FUNCTION_BLOCK FB_EQ2HOR2
VAR_INPUT
	// right ascension in degrees
	alpha: LREAL;
	// declination in degrees
	delta: LREAL;
	// longitude in degrees
	lon: LREAL;
	// latitude in degrees
	lat: LREAL;
	// Julian Days
	JD: LREAL;
END_VAR
VAR_OUTPUT
	// altitude in degrees
	alt: LREAL;
	// azimuth in degrees
	az: LREAL;
	// hour angle in degreesss
	ha: LREAL;
END_VAR
VAR
	lst: LREAL;
	// helper variables
	sinalt, sinaz, cosaz, cosalt, az1, az2, az3, length,
	// in radians
	phi_r, tau_r, alpha_r, delta_r: LREAL;
	// current epoch
	J_now: 		LREAL;
	// enable precession
	precess: 	BOOL := TRUE;
	// precession function block
	fbprecess: 	FB_PRECESS;
	//precessed coordinates
	alpha1, delta1:	LREAL;
END_VAR
VAR CONSTANT
	d2r:	LREAL := PI/180.0;
	r2d:	LREAL := 180.0/PI;
	//h2r:	LREAL := PI/12.0;
	//h2d:	LREAL := 15.0;
END_VAR

(* 
source: http://star-www.st-and.ac.uk/~fv/webnotes/chapter7.htm
https://squarewidget.com/astronomical-calculations-sidereal-time/

*)
lst := ct2lst(lon, jd) * 15.0; // lst in degrees

J_now := (JD - 2451545.0)/365.25 + 2000.0; // compute current equinox
IF precess THEN
	fbprecess( ra := alpha, dec := delta, 
	EQUINOX1 := 2000.0, EQUINOX2 := J_now, 
	ra_precessed =>alpha1, dec_precessed => delta1);
ELSE
	alpha1 := alpha;
	delta1 := delta;	
END_IF

ha := MODABS(lst - alpha1, 360.0);

alpha_r := alpha1 * d2r;
delta_r := delta1 * d2r;
tau_r := lst*d2r - alpha_r;
//tau_r := MODABS(lst*d2r - alpha_r, 2.0*PI);
phi_r := lat*d2r;

//sinalt := (SIN(delta*d2r)*SIN(lat*d2r)) + (COS(delta*d2r)*COS(lat*d2r)*COS(ha*d2r));
sinalt := SIN(phi_r)*SIN(delta_r) + COS(phi_r)*COS(delta_r)*COS(tau_r);
alt := ASIN(sinalt) * r2d;
cosalt := COS(alt*d2r);

IF ABS(cosalt) > 0.0 THEN
	sinaz := -SIN(tau_r)*COS(delta_r)/cosalt;
ELSE
	sinaz := 0.0;
END_IF

IF ABS(cosalt*COS(phi_r)) > 0.0 THEN
	cosaz := (SIN(delta_r) - SIN(phi_r)*sinalt)
			/(cosalt*COS(phi_r));
ELSE
	cosaz := 0.0;
END_IF

length := sinaz*sinaz + cosaz*cosaz;

az1 := ASIN(LIMIT(-1.0, sinaz, 1.0)) * r2d;

az2 := ACOS(LIMIT(-1.0, cosaz, 1.0)) * r2d;

az3 := -ATAN2(SIN(tau_r), SIN(phi_r)*COS(tau_r) - COS(phi_r)*TAN(delta_r)) * r2d;

IF sinaz >= 0.0 AND cosaz >=0.0 THEN // Q I
	az := az1;
ELSIF sinaz < 0.0 AND cosaz >= 0.0 THEN // Q II
	az := MODABS(-az2, 360.0);
ELSIF sinaz < 0.0 AND cosaz < 0.0 THEN // Q III
	az := 180 - az1;
ELSIF sinaz >= 0.0 AND cosaz < 0.0 THEN // Q IV
	az := az2;
END_IF

END_FUNCTION_BLOCK

(* stored: Version 1.1.0.1, ProductVersion 3.1.4024.9
   POU FB_EQ2HOR2: Id {7b34f02a-1435-4300-8153-5c49f62d1b5b}, SpecialFunc None *)
